FUNCTION_BLOCK T_MonitoredValue
VAR_INPUT
END_VAR
VAR_OUTPUT
END_VAR
VAR
    _Value   : LREAL;
    _Changed : BOOL;
	_ChangeThreshold : LREAL;
END_VAR

PROPERTY Changed : BOOL
GET
Changed := _Changed;
END_GET
END_PROPERTY

METHOD Read : LREAL
VAR_INPUT
END_VAR
Read     := _Value;
_Changed := FALSE;
END_METHOD

METHOD Update
VAR_INPUT
	Value : LREAL;
END_VAR
IF ABS(Value - _Value) > _ChangeThreshold THEN
	_Value := Value;
	_Changed := TRUE;
END_IF
END_METHOD

END_FUNCTION_BLOCK

(* stored: Version 1.1.0.1, ProductVersion 3.1.4024.12
   POU T_MonitoredValue: Id {176a7684-e463-449f-a645-00e1adf47c17}, SpecialFunc None
   Folder Methods: Id {9d7daf15-32d3-484d-aa50-46e7e98e537b}
   Folder Properties: Id {46405c05-c04c-40a5-b4f3-e616aa977296}
   Property Changed: Id {bccaf053-3640-497b-9968-4d59c32e1fac}
   Get Get: Id {fb7f9c56-1c7d-4b95-9fd3-fac752216ac8}
   Method Read: Id {2fa24f69-75b6-4b6d-b9ee-b5b8f70b1cdf}
   Method Update: Id {45360995-2377-48bf-8b8b-f29587acf793} *)
